Fanuc KAREL source: kt00888.KL

PROGRAM KT00888
%STACKSIZE=65535
%PRIORITY=65535
%NOLOCKGROUP
VAR
P1 : POSITION
P2 : POSITION
OUT : POSITION
BEGIN
-- UNRESOLVED_PC line 8 opcodes [27 22 1C 76 7E 4A] marker_code=0
END KT00888
